% RSLogix 500 project project2.RSS, saved by version 8.30.00.16 %
PROJECT "UNTITLED"    % processor: Bul.1763 MicroLogix 1100 Series B %

PROGRAM FILES
  LAD 2 "MAIN"  3 rungs
  LAD 3 "DIGITAL IO"  8 rungs
  LAD 4 "CONTROLS"  15 rungs

DATA FILES
  O0 OUTPUT  5 elements
  I1 INPUT  7 elements
  S2 STATUS  66 elements
  B3 BINARY  2 elements
  T4 TIMER  5 elements
  C5 COUNTER  1 elements
  R6 CONTROL  1 elements
  N7 INTEGER  1 elements
  F8 FLOAT  1 elements

LADDER 2 "MAIN"
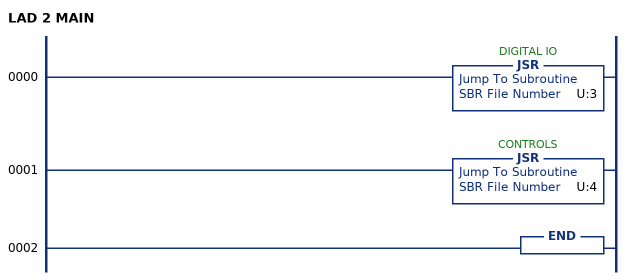
% Rung: 0 %
SOR JSR U:3 EOR
%   U:3  "DIGITAL IO" %
% Rung: 1 %
SOR JSR U:4 EOR
%   U:4  "CONTROLS" %
% Rung: 2 %
SOR END EOR

LADDER 3 "DIGITAL IO"
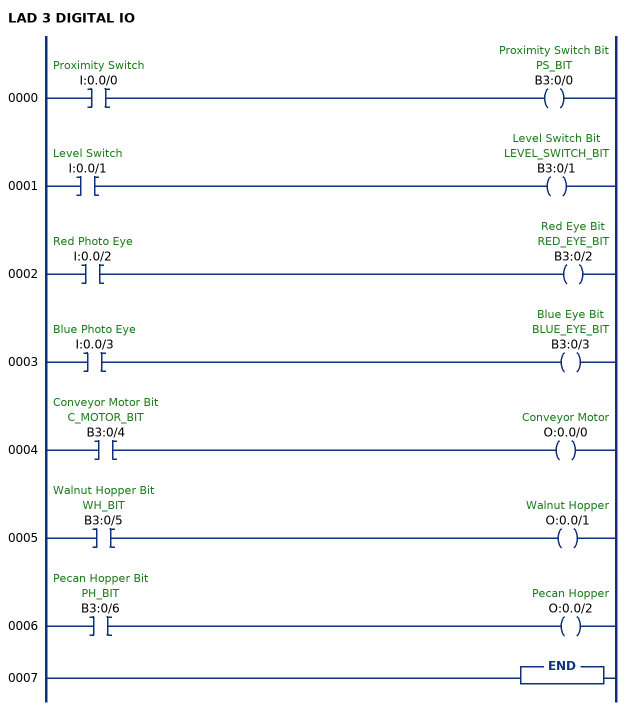
% Rung: 0 %
SOR XIC I:0.0/0 OTE B3:0/0 EOR
%   I:0.0/0  "Proximity Switch" %
%   B3:0/0  PS_BIT  "Proximity Switch Bit" %
% Rung: 1 %
SOR XIC I:0.0/1 OTE B3:0/1 EOR
%   I:0.0/1  "Level Switch" %
%   B3:0/1  LEVEL_SWITCH_BIT  "Level Switch Bit" %
% Rung: 2 %
SOR XIC I:0.0/2 OTE B3:0/2 EOR
%   I:0.0/2  "Red Photo Eye" %
%   B3:0/2  RED_EYE_BIT  "Red Eye Bit" %
% Rung: 3 %
SOR XIC I:0.0/3 OTE B3:0/3 EOR
%   I:0.0/3  "Blue Photo Eye" %
%   B3:0/3  BLUE_EYE_BIT  "Blue Eye Bit" %
% Rung: 4 %
SOR XIC B3:0/4 OTE O:0.0/0 EOR
%   B3:0/4  C_MOTOR_BIT  "Conveyor Motor Bit" %
%   O:0.0/0  "Conveyor Motor" %
% Rung: 5 %
SOR XIC B3:0/5 OTE O:0.0/1 EOR
%   B3:0/5  WH_BIT  "Walnut Hopper Bit" %
%   O:0.0/1  "Walnut Hopper" %
% Rung: 6 %
SOR XIC B3:0/6 OTE O:0.0/2 EOR
%   B3:0/6  PH_BIT  "Pecan Hopper Bit" %
%   O:0.0/2  "Pecan Hopper" %
% Rung: 7 %
SOR END EOR

LADDER 4 "CONTROLS"
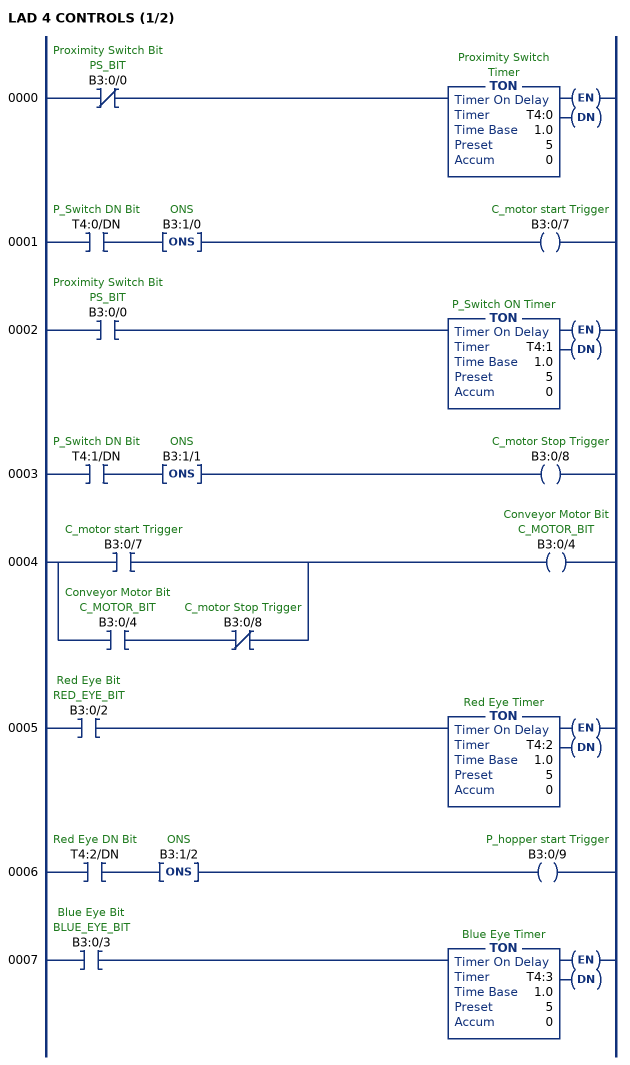
% Rung: 0 %
SOR XIO B3:0/0 TON T4:0 1.0 5 0 EOR
%   B3:0/0  PS_BIT  "Proximity Switch Bit" %
%   T4:0  "Proximity Switch Timer" %
% Rung: 1 %
SOR XIC T4:0/DN ONS B3:1/0 OTE B3:0/7 EOR
%   T4:0/DN  "P_Switch DN Bit" %
%   B3:1/0  "ONS" %
%   B3:0/7  "C_motor start Trigger" %
% Rung: 2 %
SOR XIC B3:0/0 TON T4:1 1.0 5 0 EOR
%   B3:0/0  PS_BIT  "Proximity Switch Bit" %
%   T4:1  "P_Switch ON Timer" %
% Rung: 3 %
SOR XIC T4:1/DN ONS B3:1/1 OTE B3:0/8 EOR
%   T4:1/DN  "P_Switch DN Bit" %
%   B3:1/1  "ONS" %
%   B3:0/8  "C_motor Stop Trigger" %
% Rung: 4 %
SOR BST XIC B3:0/7 NXB XIC B3:0/4 XIO B3:0/8 BND OTE B3:0/4 EOR
%   B3:0/7  "C_motor start Trigger" %
%   B3:0/4  C_MOTOR_BIT  "Conveyor Motor Bit" %
%   B3:0/8  "C_motor Stop Trigger" %
% Rung: 5 %
SOR XIC B3:0/2 TON T4:2 1.0 5 0 EOR
%   B3:0/2  RED_EYE_BIT  "Red Eye Bit" %
%   T4:2  "Red Eye Timer" %
% Rung: 6 %
SOR XIC T4:2/DN ONS B3:1/2 OTE B3:0/9 EOR
%   T4:2/DN  "Red Eye DN Bit" %
%   B3:1/2  "ONS" %
%   B3:0/9  "P_hopper start Trigger" %
% Rung: 7 %
SOR XIC B3:0/3 TON T4:3 1.0 5 0 EOR
%   B3:0/3  BLUE_EYE_BIT  "Blue Eye Bit" %
%   T4:3  "Blue Eye Timer" %

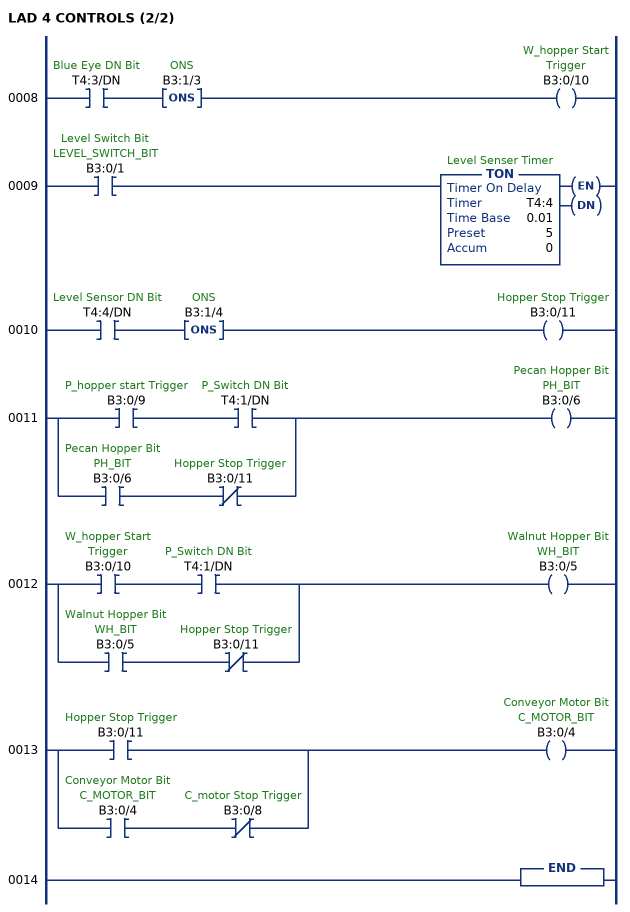
% Rung: 8 %
SOR XIC T4:3/DN ONS B3:1/3 OTE B3:0/10 EOR
%   T4:3/DN  "Blue Eye DN Bit" %
%   B3:1/3  "ONS" %
%   B3:0/10  "W_hopper Start Trigger" %
% Rung: 9 %
SOR XIC B3:0/1 TON T4:4 0.01 5 0 EOR
%   B3:0/1  LEVEL_SWITCH_BIT  "Level Switch Bit" %
%   T4:4  "Level Senser Timer" %
% Rung: 10 %
SOR XIC T4:4/DN ONS B3:1/4 OTE B3:0/11 EOR
%   T4:4/DN  "Level Sensor DN Bit" %
%   B3:1/4  "ONS" %
%   B3:0/11  "Hopper Stop Trigger" %
% Rung: 11 %
SOR BST XIC B3:0/9 XIC T4:1/DN NXB XIC B3:0/6 XIO B3:0/11 BND OTE B3:0/6 EOR
%   B3:0/9  "P_hopper start Trigger" %
%   T4:1/DN  "P_Switch DN Bit" %
%   B3:0/6  PH_BIT  "Pecan Hopper Bit" %
%   B3:0/11  "Hopper Stop Trigger" %
% Rung: 12 %
SOR BST XIC B3:0/10 XIC T4:1/DN NXB XIC B3:0/5 XIO B3:0/11 BND OTE B3:0/5 EOR
%   B3:0/10  "W_hopper Start Trigger" %
%   T4:1/DN  "P_Switch DN Bit" %
%   B3:0/5  WH_BIT  "Walnut Hopper Bit" %
%   B3:0/11  "Hopper Stop Trigger" %
% Rung: 13 %
SOR BST XIC B3:0/11 NXB XIC B3:0/4 XIO B3:0/8 BND OTE B3:0/4 EOR
%   B3:0/11  "Hopper Stop Trigger" %
%   B3:0/4  C_MOTOR_BIT  "Conveyor Motor Bit" %
%   B3:0/8  "C_motor Stop Trigger" %
% Rung: 14 %
SOR END EOR

DATA TABLE (non-zero values as saved)
DATA T4
% .PRE .ACC %
% T4:0 % 5 0
% T4:1 % 5 0
% T4:2 % 5 0
% T4:3 % 5 0
% T4:4 % 5 0
